INTERFACE I_ExtensionAddedEvent EXTENDS I_Event

PROPERTY PUBLIC TargetExtension : I_Extension
GET
END_GET
END_PROPERTY

END_INTERFACE

(* stored: Version 1.1.0.1, ProductVersion 3.1.4024.12
   Itf I_ExtensionAddedEvent: Id {15d72682-e9fd-0e9e-24b9-f648d0a1d5c4}
   Property TargetExtension: Id {cd72f87b-7f5f-025b-1dd9-dcc46f2e10aa}
   Get Get: Id {003fb858-4973-0645-35d1-0c6a8b1b6236} *)
